// TIA Portal V15.1 export
// export: Created 2024-06-21T08:41:08.5538157Z, ExportSetting WithDefaults, DisplayName Totally Integrated Automation Portal, DisplayVersion V15.1 Update 5, DisplayName TIA Portal Openness, DisplayVersion V15.1 Update 5, DisplayName SINAMICS Startdrive Advanced, DisplayVersion V15.1, DisplayName G130, G150, S120, S150, SINAMICS MV, S210, DisplayVersion V15.1, DisplayName G110M, G120, G120C, G120D, G120P, DisplayVersion V15.1, DisplayName STEP 7 Professional, DisplayVersion V15.1 Update 5, DisplayName STEP 7 Safety, DisplayVersion V15.1, DisplayName WinCC Professional, DisplayVersion V15.1 Update 5, DisplayName SIMATIC Visualization Architect, DisplayVersion V15.1
FUNCTION "LGBMotorIAnim" : Void   // FC6625, FBD
TITLE = LIAnimDWord / LGBMotorIAnim
{ S7_Optimized_Access := 'TRUE' }
AUTHOR : VCC
FAMILY : Anim
NAME : SIAnim
VERSION : 0.1
// =============================================================================
// Handles the conversion from bits to one Word for simple icon Animation. 
// =============================================================================
// stored: AutoNumber false, IsIECCheckEnabled false, SetENOAutomatically False, UDAEnableTagReadback false
   VAR_INPUT
      I_SetPos : Bool;   // Set position / Set Position
      I_Active : Bool;   // Active
      I_ManualMode : Bool;   // Manual mode / Manual Mode
      I_FncSelInHMI : Bool;   // Manual selection from HMI
      I_AlarmA : Bool;   // AlarmA
      I_AlarmB : Bool;   // AlarmB
      I_AlarmC : Bool;   // AlarmC
      I_AlarmD : Bool;   // AlarmD
      I_SafetyOk : Bool;   // Safety Ok
      I_MotionStopNok : Bool;   // Service Active / Motion stop Nok
   END_VAR
   VAR_OUTPUT
      H_IAnim : DWord;   // Icon animation Word / Icon Animation
   END_VAR
BEGIN

REGION Network 1: Icon animation Word / **** 1 - Inputs **** Set position
   // Set Position
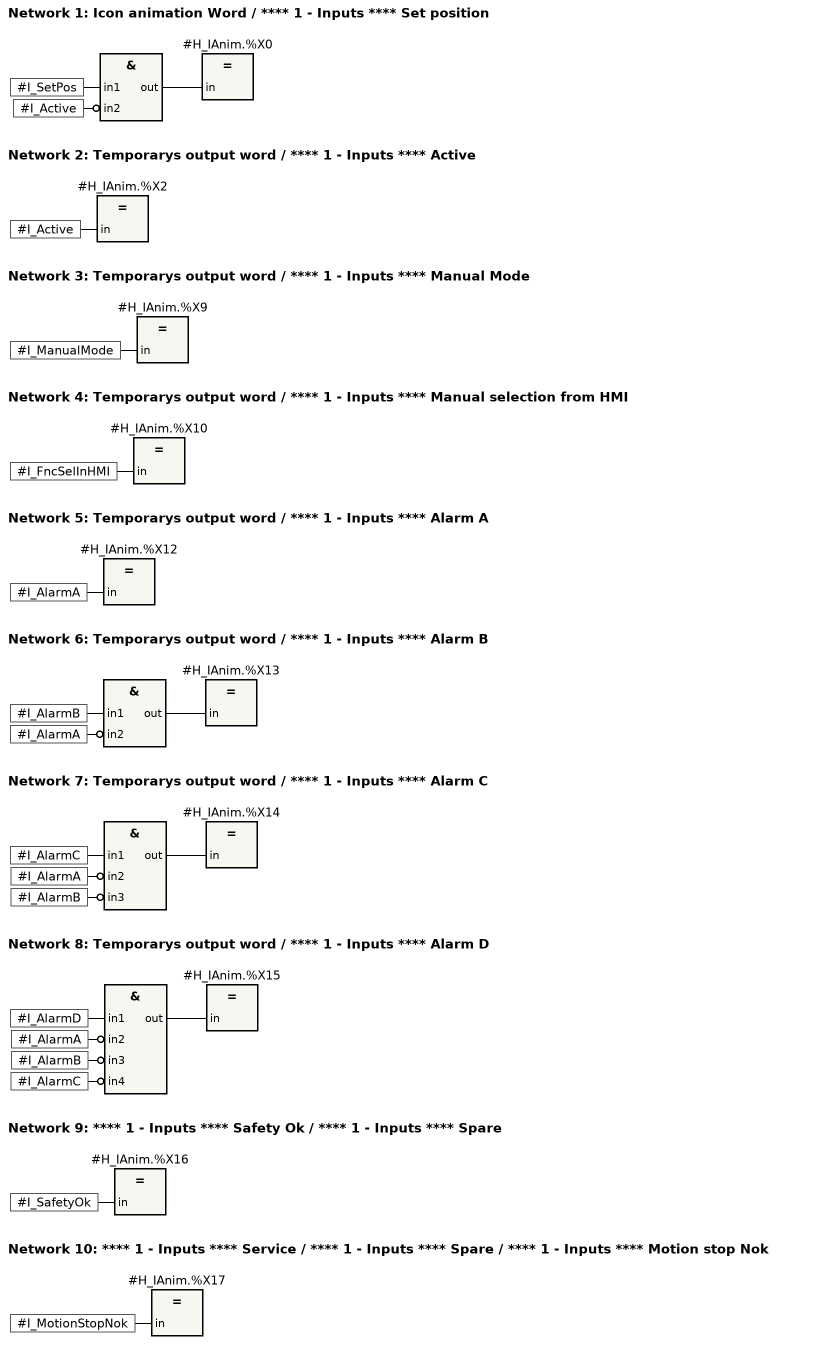
   #H_IAnim.%X0 := #I_SetPos AND NOT #I_Active;
END_REGION

REGION Network 2: Temporarys output word / **** 1 - Inputs **** Active
   // Active
   #H_IAnim.%X2 := #I_Active;
END_REGION

REGION Network 3: Temporarys output word / **** 1 - Inputs **** Manual Mode
   // Manual Mode
   #H_IAnim.%X9 := #I_ManualMode;
END_REGION

REGION Network 4: Temporarys output word / **** 1 - Inputs **** Manual selection from HMI
   // Manual selection from HMI
   #H_IAnim.%X10 := #I_FncSelInHMI;
END_REGION

REGION Network 5: Temporarys output word / **** 1 - Inputs **** Alarm A
   // Alarm A
   #H_IAnim.%X12 := #I_AlarmA;
END_REGION

REGION Network 6: Temporarys output word / **** 1 - Inputs **** Alarm B
   // Alarm B
   #H_IAnim.%X13 := #I_AlarmB AND NOT #I_AlarmA;
END_REGION

REGION Network 7: Temporarys output word / **** 1 - Inputs **** Alarm C
   // Alarm C
   #H_IAnim.%X14 := #I_AlarmC AND NOT #I_AlarmA AND NOT #I_AlarmB;
END_REGION

REGION Network 8: Temporarys output word / **** 1 - Inputs **** Alarm D
   // Alarm D
   #H_IAnim.%X15 := #I_AlarmD AND NOT #I_AlarmA AND NOT #I_AlarmB AND NOT #I_AlarmC;
END_REGION

REGION Network 9: **** 1 - Inputs **** Safety Ok / **** 1 - Inputs **** Spare
   // Safety Ok / Spare
   #H_IAnim.%X16 := #I_SafetyOk;
END_REGION

REGION Network 10: **** 1 - Inputs **** Service / **** 1 - Inputs **** Spare / **** 1 - Inputs **** Motion stop Nok
   // Service / Spare / Motion stop OK
   #H_IAnim.%X17 := #I_MotionStopNok;
END_REGION
END_FUNCTION
